FUNCTION_BLOCK CompositeBlockWithoutConnections
  FBS
    BaseBlock1 : BaseBlock;
    EA_RightPublishSubscribeAdapter_1 : EA_RightPublishSubscribeAdapter_1;
    Publish_Right_EA_1 : PUBLISH_5;
    Subscribe_Right_EA_1 : SUBSCRIBE_5;
    EA_network2_1 : EA_network2;
  END_FBS
  EVENT_CONNECTIONS
    EA_RightPublishSubscribeAdapter_1.REQ TO Publish_Right_EA_1.REQ;
    Subscribe_Right_EA_1.IND TO EA_RightPublishSubscribeAdapter_1.IND;
  END_CONNECTIONS
  DATA_CONNECTIONS
    EA_RightPublishSubscribeAdapter_1.I_E_number TO Publish_Right_EA_1.SD_1;
    EA_RightPublishSubscribeAdapter_1.I_data1 TO Publish_Right_EA_1.SD_2;
    EA_RightPublishSubscribeAdapter_1.I_data2 TO Publish_Right_EA_1.SD_3;
    EA_RightPublishSubscribeAdapter_1.N_O_data1 TO Publish_Right_EA_1.SD_4;
    EA_RightPublishSubscribeAdapter_1.N_O_data2 TO Publish_Right_EA_1.SD_5;
    Subscribe_Right_EA_1.RD_1 TO EA_RightPublishSubscribeAdapter_1.O_E_number;
    Subscribe_Right_EA_1.RD_2 TO EA_RightPublishSubscribeAdapter_1.O_data1;
    Subscribe_Right_EA_1.RD_3 TO EA_RightPublishSubscribeAdapter_1.O_data2;
    Subscribe_Right_EA_1.RD_4 TO EA_RightPublishSubscribeAdapter_1.N_I_data1;
    Subscribe_Right_EA_1.RD_5 TO EA_RightPublishSubscribeAdapter_1.N_I_data2;
  END_CONNECTIONS
  ADAPTER_CONNECTIONS
    EA_RightPublishSubscribeAdapter_1.plug TO EA_network2_1.Socket_Connection;
    EA_network2_1.Plug_Connection TO BaseBlock1.socket;
  END_CONNECTIONS
END_FUNCTION_BLOCK
